(* IEC 61131-3 sources: mect_apps/AnyTPAC/ModbusTCPserver_PLC, 4 files *)

(* ---- Resource1.gvl ---- *)
(* Global variable file *)
VAR_GLOBAL

END_VAR

(* ---- ServerTCP.gvl ---- *)
(*Global variable file*)
(*[[
]]*)

VAR_GLOBAL

	(* PLC_time AT %MD0.21560:REAL; *)		PLC_time_LO		AT %MW0.21560:WORD;	PLC_time_HI		AT %MW0.21562:WORD;
	(* PLC_timeMin AT %MD0.21564:REAL; *)	PLC_timeMin_LO	AT %MW0.21564:WORD;	PLC_timeMin_HI	AT %MW0.21566:WORD;
	(* PLC_timeMax AT %MD0.21568:REAL; *)	PLC_timeMax_LO	AT %MW0.21568:WORD;	PLC_timeMax_HI	AT %MW0.21570:WORD;

	I_DigitalOutput_1 AT %IW4.0 : INT; (* BOOL *)
	I_DigitalOutput_2 AT %IW4.2 : INT; (* BOOL *)
	I_DigitalInput_3  AT %IW4.4 : INT; (* BOOL *)
	I_DigitalInput_4  AT %IW4.6 : INT; (* BOOL *)
	I_TimeValue_LO    AT %IW4.8 : WORD; (* REAL *)
	I_TimeValue_HI    AT %IW4.10 : WORD;
	I_TimeMin_LO      AT %IW4.12 : WORD; (* REAL *)
	I_TimeMin_HI      AT %IW4.14 : WORD;
	I_TimeMax_LO      AT %IW4.16 : WORD; (* REAL *)
	I_TimeMax_HI      AT %IW4.18 : WORD;
	I_AnalogInput_1   AT %IW4.20 : INT; (* INT.3 *)
	I_AnalogInput_2   AT %IW4.22 : INT; (* INT.1 *)
	(* ... *)
	I_HOLDING_4095    AT %IW4.8190: UINT;

	Q_DigitalOutput_1 AT %QW4.0 : INT; (* BOOL *)
	Q_DigitalOutput_2 AT %QW4.2 : INT; (* BOOL *)
	Q_DigitalInput_3  AT %QW4.4 : INT; (* BOOL *)
	Q_DigitalInput_4  AT %QW4.6 : INT; (* BOOL *)
	Q_TimeValue_LO    AT %QW4.8 : WORD; (* REAL *)
	Q_TimeValue_HI    AT %QW4.10 : WORD;
	Q_TimeMin_LO      AT %QW4.12 : WORD; (* REAL *)
	Q_TimeMin_HI      AT %QW4.14 : WORD;
	Q_TimeMax_LO      AT %QW4.16 : WORD; (* REAL *)
	Q_TimeMax_HI      AT %QW4.18 : WORD;
	Q_AnalogInput_1   AT %QW4.20 : INT; (* INT.3 *)
	Q_AnalogInput_2   AT %QW4.22 : INT; (* INT.1 *)
	(* ... *)
	Q_HOLDING_4095    AT %QW4.8190: UINT;

END_VAR

(* ---- fb_HW119_Check.st ---- *)
(*[[
]]*)
FUNCTION_BLOCK fb_HW119_Check
#import "Resource1.gvl"
#import "crosstable.gvl"
VAR_INPUT
END_VAR
VAR
	STATE:UINT;
	FunctRes:UINT;
	TON_Reconnect:TON;
	InitCommunication:fb_HW119_InitComm;

END_VAR

		TON_Reconnect(IN := TRUE,PT := T#4s);

		IF TON_Reconnect.Q 	THEN
			CASE STATE OF
				10: STATE:=20;
				20:	STATE:=30;
				30:	STATE:=10;
			ELSE
				STATE:=10;
			END_CASE;
		END_IF;

		IF NOT RTU_RUN AND RTUProtocol_ON AND STATE = 10 AND TON_Reconnect.Q THEN
			InitCommunication(ENABLE:=TRUE,Interface:='RTU');	(*inizializza comunicazione	*)
			IF InitCommunication.END THEN
				FunctRes:=WORD_TO_UINT(TSK_Start('TASK2_RTU'));		(* partenza task RTU*)
				InitCommunication(ENABLE:=FALSE);
				STATE:=20;
				RTU_RUN:=TRUE;
				TON_Reconnect(In:=FALSE);
			ELSIF InitCommunication.ERR THEN
				TON_Reconnect(In:=FALSE);
				InitCommunication(ENABLE:=FALSE);
				RTU_RUN:=FALSE;
				STATE:=20;
			END_IF;
		ELSIF NOT TCP_RUN AND TCPProtocol_ON AND STATE = 20 AND TON_Reconnect.Q 	THEN
			InitCommunication(ENABLE:=TRUE,Interface:='TCP');	(*inizializza comunicazione	*)
			IF InitCommunication.END THEN
				FunctRes:=WORD_TO_UINT(TSK_Start('TASK3_TCP'));		(* partenza task TCP*)
				InitCommunication(ENABLE:=FALSE);
				STATE:=30;
				TCP_RUN:=TRUE;
				TON_Reconnect(In:=FALSE);
			ELSIF InitCommunication.ERR THEN
				TON_Reconnect(In:=FALSE);
				InitCommunication(ENABLE:=FALSE);
				TCP_RUN:=FALSE;
				STATE:=30;
			END_IF;
		ELSIF NOT TCPRTU_RUN AND TCPRTUProtocol_ON AND STATE = 30	AND TON_Reconnect.Q 	 	THEN
			TON_Reconnect(In:=FALSE);
			InitCommunication(ENABLE:=TRUE,Interface:='TCPRTU');	(*inizializza comunicazione	*)
			IF InitCommunication.END THEN
				FunctRes:=WORD_TO_UINT(TSK_Start('TASK4_TCPRTU'));		(* partenza task TCPRTU*)
				InitCommunication(ENABLE:=FALSE);
				STATE:=10;
				TCPRTU_RUN:=TRUE;
				TON_Reconnect(In:=FALSE);
			ELSIF InitCommunication.ERR THEN
				TON_Reconnect(In:=FALSE);
				InitCommunication(ENABLE:=FALSE);
				TCPRTU_RUN:=FALSE;
				STATE:=10;

			END_IF;
		END_IF;

END_FUNCTION_BLOCK

(* ---- PLC.st ---- *)
(*[[
]]*)
PROGRAM PLC
#import "Resource1.gvl"
#import "TPACLocaIO.gvl"
#import "ServerTCP.gvl"
VAR
	info : TSK_INFO ;
	counter : INT := 0;
	task_ms : INT := -1;
	square_ms : INT := 1000;
	retval : WORD;
	first : BOOL := true;
END_VAR;
	if first then
		first := false;
		if task_ms < 0 then
			retval := TSK_GetInfo('Task0_Control', info);
			task_ms := TIME_TO_INT(info.tCycle);
		end_if;
	end_if;

	counter := (counter + 1) mod 10000;

	(* Input Simulation *)
	PLC_DigIn_1 := PLC_DigOut_1;
	PLC_DigIn_2 := PLC_DigOut_2;
	PLC_DigIn_3 := PLC_DigOut_3;
	PLC_DigIn_4 := PLC_DigOut_4;
	PLC_DigIn_5 := PLC_DigOut_5;
	PLC_DigIn_6 := PLC_DigOut_6;
	PLC_DigIn_7 := PLC_DigOut_7;
	PLC_DigIn_8 := PLC_DigOut_8;
	PLC_AnIn_1 := 5000 + REAL_TO_INT(5000.0 * sin(PLC_time / 1.0));
	PLC_AnIn_2 := 10000 * WORD_TO_INT(PLC_DigOut_1);

	(* Output Simulation *)
	if (REAL_TO_INT(PLC_time) mod 2) = 0 then
		PLC_DigOut_1 := 1;
		PLC_DigOut_2 := 0;
		PLC_DigOut_3 := 1;
		PLC_DigOut_4 := 0;
		PLC_DigOut_5 := 0;
		PLC_DigOut_6 := 1;
		PLC_DigOut_7 := 0;
		PLC_DigOut_8 := 1;
	else
		PLC_DigOut_1 := 0;
		PLC_DigOut_2 := 1;
		PLC_DigOut_3 := 0;
		PLC_DigOut_4 := 1;
		PLC_DigOut_5 := 1;
		PLC_DigOut_6 := 0;
		PLC_DigOut_7 := 1;
		PLC_DigOut_8 := 0;
	end_if;

	(* Modbus TCP Server *)
	Q_DigitalOutput_1 := WORD_TO_INT(PLC_DigIn_1);
	Q_DigitalOutput_2 := WORD_TO_INT(PLC_DigIn_2);
	Q_DigitalInput_3 := WORD_TO_INT(PLC_DigIn_3);
	Q_DigitalInput_4 := WORD_TO_INT(PLC_DigIn_4);
	Q_TimeValue_LO := PLC_time_LO;
	Q_TimeValue_HI := PLC_time_HI;
	Q_TimeMin_LO := PLC_timeMin_LO;
	Q_TimeMin_HI := PLC_timeMin_HI;
	Q_TimeMax_LO := PLC_timeMax_LO;
	Q_TimeMax_HI := PLC_timeMax_HI;
	Q_AnalogInput_1 := PLC_AnIn_1;
	Q_AnalogInput_2 := PLC_AnIn_2;

END_PROGRAM
